TYPE ST_SmokeDetectors :
STRUCT
	State : eSmokeDetectAlarmStatus;
END_STRUCT
END_TYPE

(* stored: Version 1.1.0.1, ProductVersion 3.1.4024.12
   DUT ST_SmokeDetectors: Id {7a2e078f-883e-48d0-a0b5-2f835a953f4a} *)
